Omron CX-Programmer project NuevoProyecto (CX-Programmer 9.61)

# PLC P2E1V2: CJ2M CPU11

## Program NuevoPrograma1 (cyclic task 0)
Local symbols
Amarillo1 1.01 BOOL  ; 1.01
Amarillo2 1.09 BOOL  ; 1.09
Entrada1 0.00 BOOL  ; 0.00
Entrada2 0.01 BOOL  ; 0.01
P0 2.00 BOOL  ; 2.0
P1 2.01 BOOL  ; 2.01
P2 2.02 BOOL  ; 2.02
P3 2.03 BOOL  ; 2.03
P4 2.04 BOOL  ; 2.04
P5 2.05 BOOL  ; 2.05
P6 2.06 BOOL  ; 2.06
P7 2.07 BOOL  ; 2.07
P8 2.08 BOOL  ; 2.08
P9 2.09 BOOL  ; 2.09
Rojo1 1.00 BOOL  ; 1.00
Rojo2 1.08 BOOL  ; 1.08
Verde1 1.02 BOOL  ; 1.02
Verde2 1.10 BOOL  ; 1.10

### Section Sección1

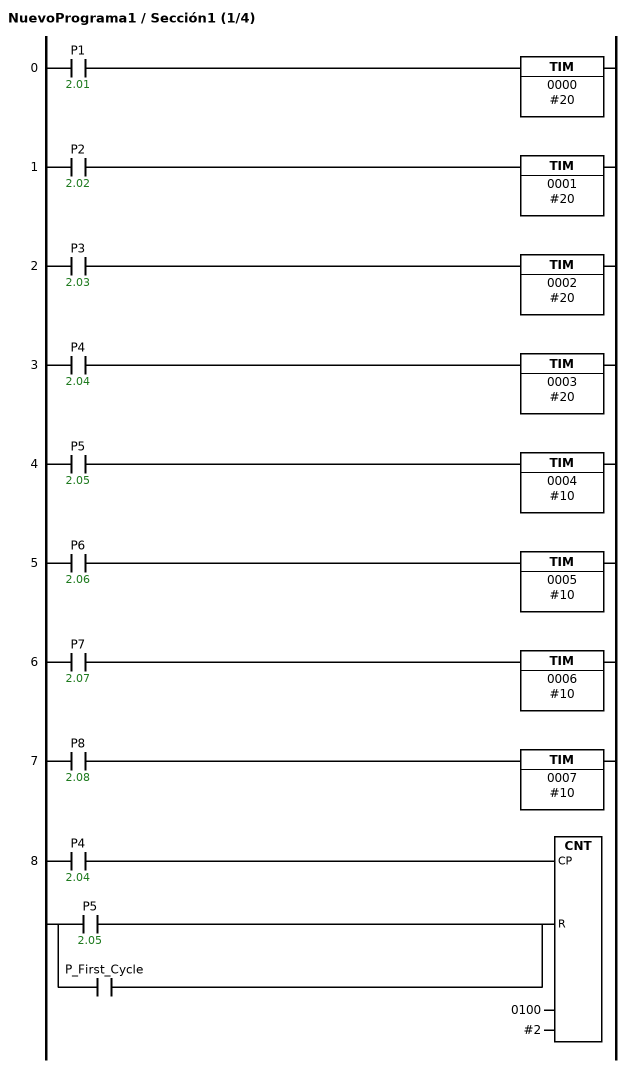
; rung 0
LD P1  ; 2.01
TIM 0000 #20
; rung 1
LD P2  ; 2.02
TIM 0001 #20
; rung 2
LD P3  ; 2.03
TIM 0002 #20
; rung 3
LD P4  ; 2.04
TIM 0003 #20
; rung 4
LD P5  ; 2.05
TIM 0004 #10
; rung 5
LD P6  ; 2.06
TIM 0005 #10
; rung 6
LD P7  ; 2.07
TIM 0006 #10
; rung 7
LD P8  ; 2.08
TIM 0007 #10
; rung 8
LD P4  ; 2.04
LD P5  ; 2.05
OR P_First_Cycle
CNT 0100 #2

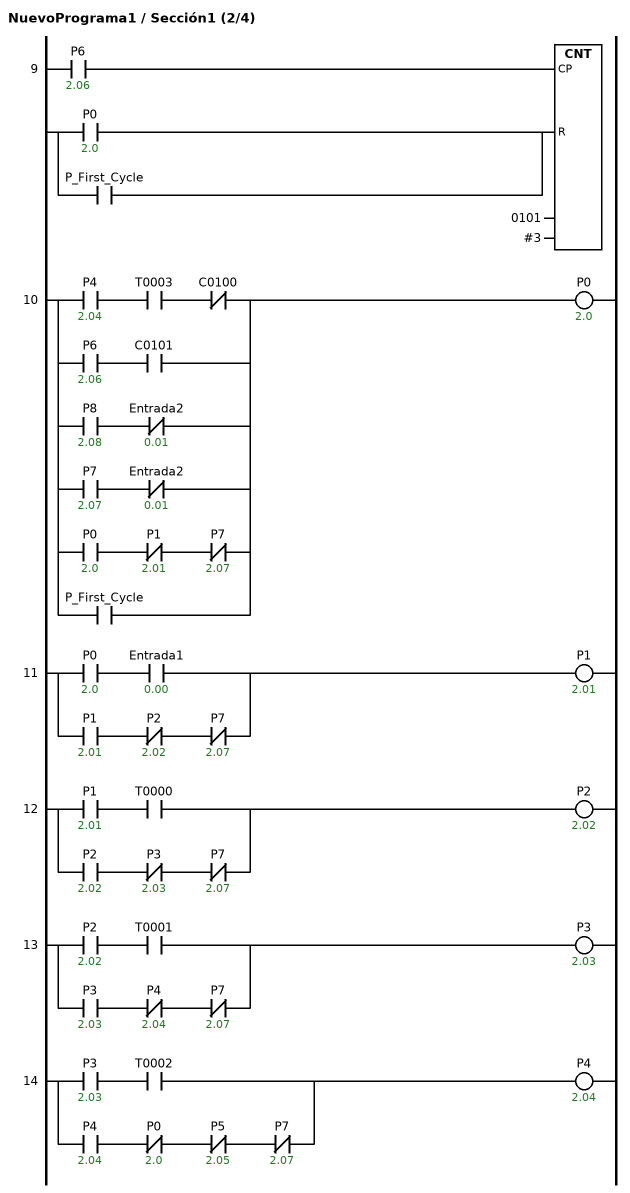
; rung 9
LD P6  ; 2.06
LD P0  ; 2.0
OR P_First_Cycle
CNT 0101 #3
; rung 10
LD P4  ; 2.04
AND T0003
ANDNOT C0100
LD P6  ; 2.06
AND C0101
ORLD
LD P8  ; 2.08
ANDNOT Entrada2  ; 0.01
ORLD
LD P7  ; 2.07
ANDNOT Entrada2  ; 0.01
ORLD
LD P0  ; 2.0
ANDNOT P1  ; 2.01
ANDNOT P7  ; 2.07
ORLD
OR P_First_Cycle
OUT P0  ; 2.0
; rung 11
LD P0  ; 2.0
AND Entrada1  ; 0.00
LD P1  ; 2.01
ANDNOT P2  ; 2.02
ANDNOT P7  ; 2.07
ORLD
OUT P1  ; 2.01
; rung 12
LD P1  ; 2.01
AND T0000
LD P2  ; 2.02
ANDNOT P3  ; 2.03
ANDNOT P7  ; 2.07
ORLD
OUT P2  ; 2.02
; rung 13
LD P2  ; 2.02
AND T0001
LD P3  ; 2.03
ANDNOT P4  ; 2.04
ANDNOT P7  ; 2.07
ORLD
OUT P3  ; 2.03
; rung 14
LD P3  ; 2.03
AND T0002
LD P4  ; 2.04
ANDNOT P0  ; 2.0
ANDNOT P5  ; 2.05
ANDNOT P7  ; 2.07
ORLD
OUT P4  ; 2.04

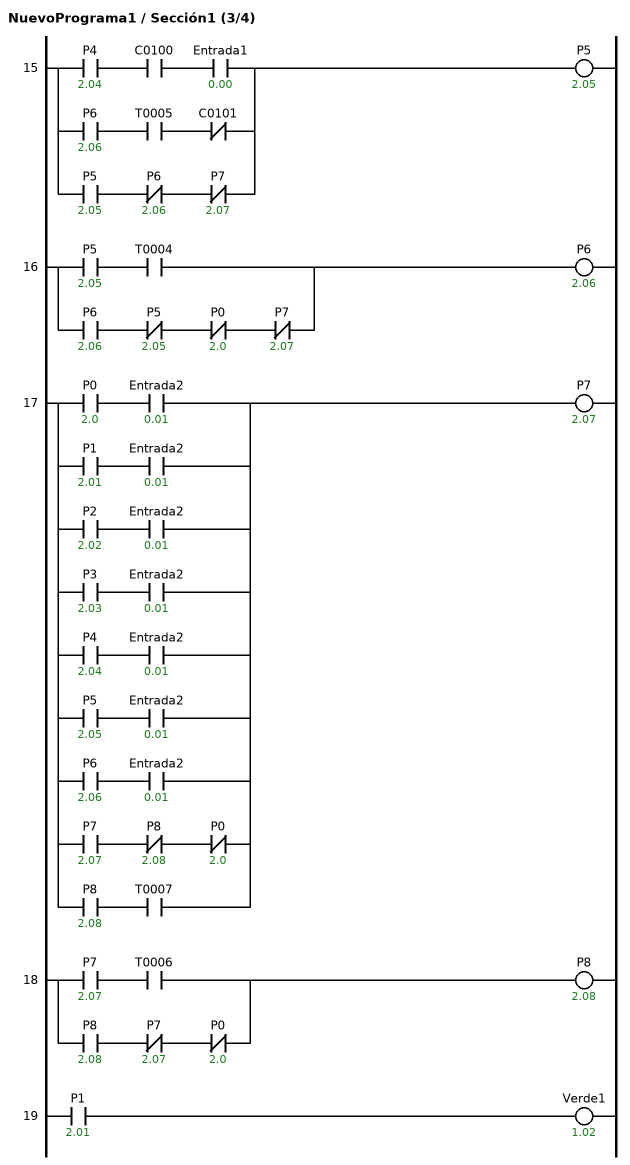
; rung 15
LD P4  ; 2.04
AND C0100
AND Entrada1  ; 0.00
LD P6  ; 2.06
AND T0005
ANDNOT C0101
ORLD
LD P5  ; 2.05
ANDNOT P6  ; 2.06
ANDNOT P7  ; 2.07
ORLD
OUT P5  ; 2.05
; rung 16
LD P5  ; 2.05
AND T0004
LD P6  ; 2.06
ANDNOT P5  ; 2.05
ANDNOT P0  ; 2.0
ANDNOT P7  ; 2.07
ORLD
OUT P6  ; 2.06
; rung 17
LD P0  ; 2.0
AND Entrada2  ; 0.01
LD P1  ; 2.01
AND Entrada2  ; 0.01
ORLD
LD P2  ; 2.02
AND Entrada2  ; 0.01
ORLD
LD P3  ; 2.03
AND Entrada2  ; 0.01
ORLD
LD P4  ; 2.04
AND Entrada2  ; 0.01
ORLD
LD P5  ; 2.05
AND Entrada2  ; 0.01
ORLD
LD P6  ; 2.06
AND Entrada2  ; 0.01
ORLD
LD P7  ; 2.07
ANDNOT P8  ; 2.08
ANDNOT P0  ; 2.0
ORLD
LD P8  ; 2.08
AND T0007
ORLD
OUT P7  ; 2.07
; rung 18
LD P7  ; 2.07
AND T0006
LD P8  ; 2.08
ANDNOT P7  ; 2.07
ANDNOT P0  ; 2.0
ORLD
OUT P8  ; 2.08
; rung 19
LD P1  ; 2.01
OUT Verde1  ; 1.02

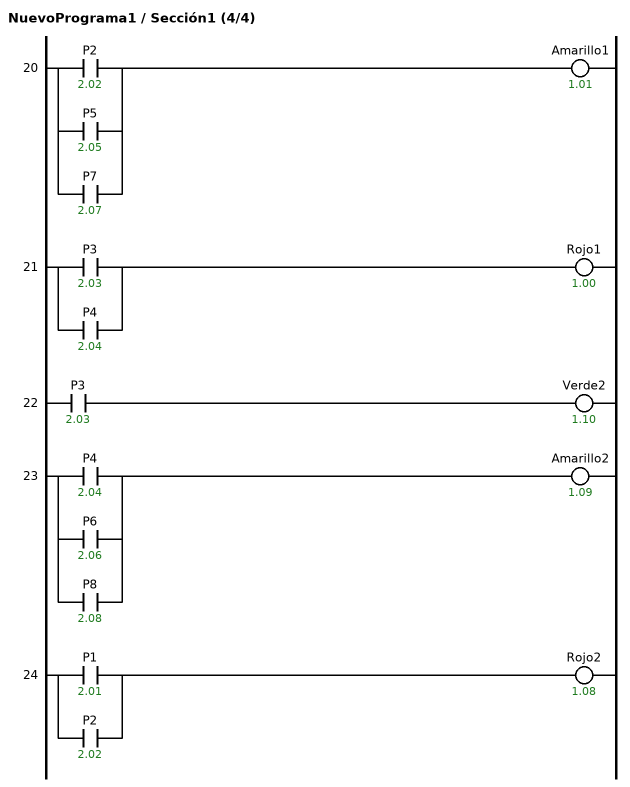
; rung 20
LD P2  ; 2.02
OR P5  ; 2.05
OR P7  ; 2.07
OUT Amarillo1  ; 1.01
; rung 21
LD P3  ; 2.03
OR P4  ; 2.04
OUT Rojo1  ; 1.00
; rung 22
LD P3  ; 2.03
OUT Verde2  ; 1.10
; rung 23
LD P4  ; 2.04
OR P6  ; 2.06
OR P8  ; 2.08
OUT Amarillo2  ; 1.09
; rung 24
LD P1  ; 2.01
OR P2  ; 2.02
OUT Rojo2  ; 1.08

### Section END
; rung 0
END(001)